FUNCTION_BLOCK FB_CTU_DINT (* Up counter *)
  (* Standard: 61499-1; Description: Copyright (c) 2023 Martin Erich Jobst This program and the accompanying materials are made available under the terms of the Eclipse Public License 2.0 which is available at https://www.eclipse.org/legal/epl-2.0/ SPDX-License-Identifier: EPL-2.0 *)
  (* Version 1.0, 2023-04-28, Martin Jobst *)
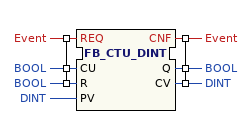
  EVENT_INPUT
    REQ WITH CU, R; (* Normal Execution Request *)
  END_EVENT
  EVENT_OUTPUT
    CNF WITH Q, CV; (* Execution Confirmation *)
  END_EVENT
  VAR_INPUT
    CU : BOOL; (* Count up *)
    R : BOOL; (* Reset *)
    PV : DINT; (* Preset value *)
  END_VAR
  VAR_OUTPUT
    Q : BOOL; (* Output *)
    CV : DINT; (* Count value *)
  END_VAR
  ALGORITHM REQ IN ST:
IF R THEN
  CV := 0;
ELSIF CU AND CV < 2147483647 THEN
  CV := CV + 1;
END_IF;
Q := CV >= PV;
  END_ALGORITHM
END_FUNCTION_BLOCK
